TYPE DUT_Switch :
STRUCT
	///////////////////////////////////////////////////////////////////////////////////////////////////////////////////////////////////////////
	// Settings
	///////////////////////////////////////////////////////////////////////////////////////////////////////////////////////////////////////////
	
	
	
	///////////////////////////////////////////////////////////////////////////////////////////////////////////////////////////////////////////
	// Status
	///////////////////////////////////////////////////////////////////////////////////////////////////////////////////////////////////////////
	
	
	
	///////////////////////////////////////////////////////////////////////////////////////////////////////////////////////////////////////////
	// Control & return
	///////////////////////////////////////////////////////////////////////////////////////////////////////////////////////////////////////////
	
	Q									: BOOL; 
	
	
	///////////////////////////////////////////////////////////////////////////////////////////////////////////////////////////////////////////
	// Mapping
	///////////////////////////////////////////////////////////////////////////////////////////////////////////////////////////////////////////
END_STRUCT
END_TYPE

(* stored: Version 1.1.0.1, ProductVersion 3.1.4022.12
   DUT DUT_Switch: Id {7fc1c06c-7ac6-430c-8fa6-fc757144cc56} *)
